FUNCTION_BLOCK FB_Discharge
VAR_INPUT
END_VAR
VAR_OUTPUT
END_VAR
VAR
END_VAR

END_FUNCTION_BLOCK

(* stored: Version 1.1.0.1
   POU FB_Discharge: Id {9b334204-e1f0-4f77-8568-487de87d10d1}, SpecialFunc None *)
